PROGRAM MAIN
VAR
	bInit : BOOL := TRUE;	
	test : LTIME_OF_DAY;
END_VAR

(* Static values and namespace test are initialized only once upon startup *)
IF bInit THEN
	bInit := FALSE;
	PRG_Static();
END_IF
PRG_Dynamic();

END_PROGRAM

(* stored: Version 1.1.0.1
   POU MAIN: Id {95eb49a5-1119-4202-a665-eb5eaccb2021}, SpecialFunc None *)
